(* Logix 5000 project; controller EuniceF_ICA14 vendor 1 type 14 code 150 rev 37.11; software revision 37.00 *)

TASK MainTask (continuous, watchdog 500 ms) : MainProgram

MODULES
   Local : vendor 1 type 14 code 150 (Compact 0, rev 37.11)
      Discrete_IO : Embedded (Compact 1, rev 3.1, Output RPI 20 ms)
      Analog_IO : Embedded (Compact 2, rev 1.1, Output RPI 80 ms)
      Counters : Embedded (Compact 3, rev 1.1, Output RPI 20 ms)
END_MODULES

VAR_GLOBAL   (* controller tags *)
   B1 : ALIAS FOR Local:1:I.Data.12;
   B2 : ALIAS FOR Local:1:I.Data.13;
   Button : ALIAS FOR Local:1:I.Data.11;
   DEL1 : TIMER := (PRE := 3000);
   DEL2 : TIMER := (PRE := 2000);
   L1 : ALIAS FOR Local:1:O.Data.2;
   L2 : ALIAS FOR Local:1:O.Data.3;
   Light : ALIAS FOR Local:1:O.Data.1;
   Seq1 : DINT;
   Seq2 : DINT;
   Timer1 : TIMER := (PRE := 2000);
END_VAR

PROGRAM MainProgram   (* main routine MainRoutine *)

ROUTINE MainRoutine   (* ladder *)
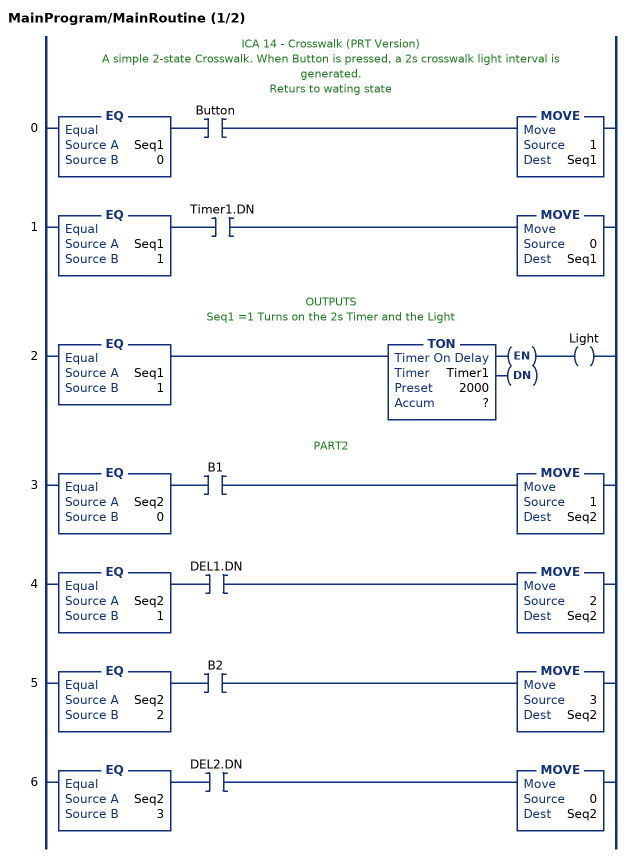
   // ICA 14 - Crosswalk (PRT Version)
   // A simple 2-state Crosswalk. When Button is pressed, a 2s crosswalk light interval is generated.
   // Returs to wating state
   0: EQ(Seq1,0)XIC(Button)MOVE(1,Seq1);
   1: EQ(Seq1,1)XIC(Timer1.DN)MOVE(0,Seq1);
   // OUTPUTS
   // Seq1 =1 Turns on the 2s Timer and the Light
   2: EQ(Seq1,1)TON(Timer1,?,?)OTE(Light);
   // PART2
   3: EQ(Seq2,0)XIC(B1)MOVE(1,Seq2);
   4: EQ(Seq2,1)XIC(DEL1.DN)MOVE(2,Seq2);
   5: EQ(Seq2,2)XIC(B2)MOVE(3,Seq2);
   6: EQ(Seq2,3)XIC(DEL2.DN)MOVE(0,Seq2);
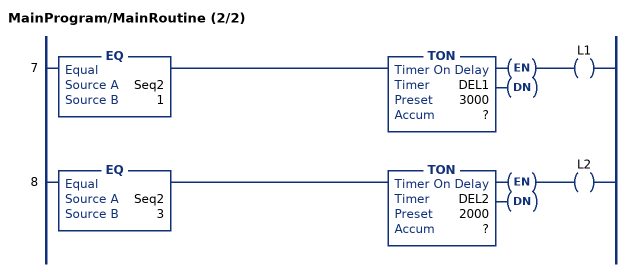
   7: EQ(Seq2,1)TON(DEL1,?,?)OTE(L1);
   8: EQ(Seq2,3)TON(DEL2,?,?)OTE(L2);
END_ROUTINE
END_PROGRAM
